(* CoDeSys 2.3.9.47 project: OR GATE.pro *)
(* Libraries: Nexgenie.lib 28.8.18 12:27:24, Standard.lib 28.8.18 12:27:25, Nexgenie_Util.lib 28.8.18 12:27:24, Nexgenie_H.lib 28.8.18 12:27:24, VAW.lib 28.8.18 12:27:25, Modbus.lib 28.8.18 12:27:24 *)

(* PLC configuration (modules and I/O channels)
Nexgenie1000 [Root] node -1, in %IB0 out %QB0
  Nexgenie [Nexgenie] node 0, in %IB0 out %QB0
*)

(* POU PLC_PRG, LD *)
PROGRAM PLC_PRG
VAR
	A AT %IX0.0: BOOL;
	B AT %IX0.1: BOOL;
	Z AT %QX0.0: BOOL;
END_VAR
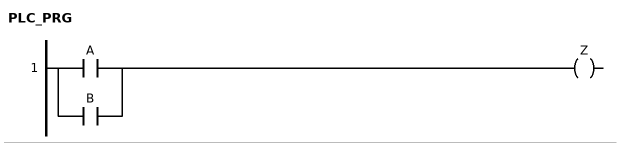
_LD_ (* Ladder Diagram *)
NETWORK 1
	{ [A] | [B] } --- (Z)
_END_LD_
(* the same logic as Structured Text *)
(* Network 1 *)
Z := A OR B;
END_PROGRAM

(* Visualisation LOL
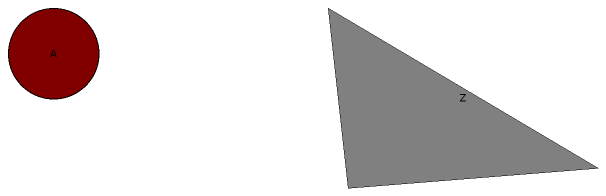
polygon at (390,70)-(660,250): text "Z"; alarm colour if PLC_PRG.Z
ellipse at (70,70)-(161,161): text "A"; alarm colour if PLC_PRG.A; toggles PLC_PRG.A
1 elements of other kinds (tables, trends, ...) not read
*)
